(* Logix 5000 project; controller PROCESS_OUTPUT Emulate 5570 rev 33.11; software revision 33.00 *)

TASK MainTask (continuous, watchdog 500 ms) : MainProgram

MODULES
   Local : Emulate 5570 (ICP 2, rev 33.11)
       : 1756-IB16 (ICP 3, rev 3.1, Input RPI 20 ms)
       : vendor 1 type 7 code 16 (ICP 4, rev 3.1, Output RPI 20 ms)
END_MODULES

VAR_GLOBAL   (* controller tags *)
   PROCESS_OUTPUT : ALIAS FOR Local:4:O.Data.0;   // Process Output
   SW_START : ALIAS FOR Local:3:I.Data.0;   // START Momentary N. O. Pushbutton
END_VAR

PROGRAM MainProgram   (* main routine MainRoutine *)
VAR
   A_MATERIAL_MULTIPLIER : REAL;   // Material A Multiplier
   B_MATERIAL_MULTIPLIER : REAL;   // Material B Multiplier
   C_MATERIAL_MULTIPLIER : REAL;   // Material C Multiplier
   D_MATERIAL_MULTIPLIER : REAL;   // Material D Multiplier
   HMI_A_MATERIAL_MULTIPLIER : ALIAS FOR A_MATERIAL_MULTIPLIER;
   HMI_ACC_PROCESS_TIME : ALIAS FOR PROCESS_TIME.ACC;
   HMI_B_MATERIAL_MULTIPLIER : ALIAS FOR B_MATERIAL_MULTIPLIER;
   HMI_C_MATERIAL_MULTIPLIER : ALIAS FOR C_MATERIAL_MULTIPLIER;
   HMI_D_MATERIAL_MULTIPLIER : ALIAS FOR D_MATERIAL_MULTIPLIER;
   HMI_NUM_SHEETS : ALIAS FOR NUM_SHEETS;
   HMI_PRE_PROCESS_TIME : ALIAS FOR PROCESS_TIME.PRE;
   HMI_TYPE_SHEET : ALIAS FOR TYPE_SHEET;
   MATERIAL_MULTI_VALUE : REAL;   // Material Multiplier Value
   NUM_SHEETS : INT;   // Value for Sheet Type
   PROCESS_TIME : TIMER;   // Process Timer
   PROCESS_VALUE : REAL;   // Process Value
   TYPE_SHEET : INT;   // Value Number of Sheets
END_VAR

ROUTINE MainRoutine   (* ladder *)
   0: ;
END_ROUTINE
END_PROGRAM
